// TIA Portal project "Bai 7" (V16)

(* hardware
DEVICE "S7-1200 station_1"  S7-1200 Station
   slot 0: "Rack_0"  S7-1200 Rack  Rack  V1.0
   slot 1: "PLC_1"  CPU 1214C DC/DC/DC  6ES7 214-1AG40-0XB0  V4.2
   slot 2: "DQ 16xRelay_1"  SM 1222 DQ16 x relay  6ES7 222-1HH32-0XB0  V2.0
*)

// ===== PLC "PLC_1"  CPU 1214C DC/DC/DC =====

VAR_GLOBAL   // PLC tag table "Default tag table"
   "Start" AT %I0.0 : Bool;
   "Quay_DC" AT %Q9.1 : Bool;
   "Khoan" AT %Q9.2 : Bool;
   "Biến giữ chương trình" AT %M0.0 : Bool;
   "SQ1" AT %I0.1 : Bool;
   "Biến giữ timer T5" AT %M1.1 : Bool;
   "Biến kích động cơ" AT %M1.2 : Bool;
   "Stop" AT %I1.0 : Bool;
   "Tag_11" AT %M1.3 : Bool;
   "Tag_12" AT %M0.1 : Bool;
   "Biến giữ quay DC" AT %M0.2 : Bool;
   "Tag_1" AT %M1.4 : Bool;
   "Tag_2" AT %M1.7 : Bool;
   "Tag_10" AT %M1.0 : Bool;
   "Biến kích nhánh 2" AT %M0.7 : Bool;
   "SQ2" AT %I0.2 : Bool;
   "SQ3" AT %I0.3 : Bool;
   "Biến giữ kẹp phôi" AT %M0.3 : Bool;
   "Biến giữ khoan" AT %M0.4 : Bool;
   "KepPhoi" AT %Q9.3 : Bool;
   "Biến giữ timer T3" AT %M0.5 : Bool;
   "Biến giữ timer T4" AT %M0.6 : Bool;
END_VAR

// folder: System blocks/Program resources

DATA_BLOCK "T1"   // DB1
{ S7_Optimized_Access := 'TRUE' }
AUTHOR : Simatic
FAMILY : IEC
NAME : IEC_TMR
VERSION : 1.0
// stored: InstanceOfName IEC_TIMER
"IEC_TIMER"
BEGIN
END_DATA_BLOCK

DATA_BLOCK "T2"   // DB2
{ S7_Optimized_Access := 'TRUE' }
AUTHOR : Simatic
FAMILY : IEC
NAME : IEC_TMR
VERSION : 1.0
// stored: InstanceOfName IEC_TIMER
"IEC_TIMER"
BEGIN
END_DATA_BLOCK

DATA_BLOCK "T3"   // DB3
{ S7_Optimized_Access := 'TRUE' }
AUTHOR : Simatic
FAMILY : IEC
NAME : IEC_TMR
VERSION : 1.0
// stored: InstanceOfName IEC_TIMER
"IEC_TIMER"
BEGIN
END_DATA_BLOCK

DATA_BLOCK "T4"   // DB4
{ S7_Optimized_Access := 'TRUE' }
AUTHOR : Simatic
FAMILY : IEC
NAME : IEC_TMR
VERSION : 1.0
// stored: InstanceOfName IEC_TIMER
"IEC_TIMER"
BEGIN
END_DATA_BLOCK

DATA_BLOCK "T5"   // DB5
{ S7_Optimized_Access := 'TRUE' }
AUTHOR : Simatic
FAMILY : IEC
NAME : IEC_TMR
VERSION : 1.0
// stored: InstanceOfName IEC_TIMER
"IEC_TIMER"
BEGIN
END_DATA_BLOCK

DATA_BLOCK "T6"   // DB6
{ S7_Optimized_Access := 'TRUE' }
AUTHOR : Simatic
FAMILY : IEC
NAME : IEC_TMR
VERSION : 1.0
// stored: InstanceOfName IEC_TIMER
"IEC_TIMER"
BEGIN
END_DATA_BLOCK

// folder: (top level)

ORGANIZATION_BLOCK "Main"   // OB1, LAD, ProgramCycle
TITLE = "Main Program Sweep (Cycle)"
{ S7_Optimized_Access := 'TRUE' }
VERSION : 0.1
   VAR_INPUT
      Initial_Call : Bool;   // Initial call of this OB
      Remanence : Bool;   // =True, if remanent data are available
   END_VAR
   VAR_TEMP   // added for the SCL form of the ladder/FBD networks
      _w1 : Bool;
   END_VAR
BEGIN

REGION Network 1
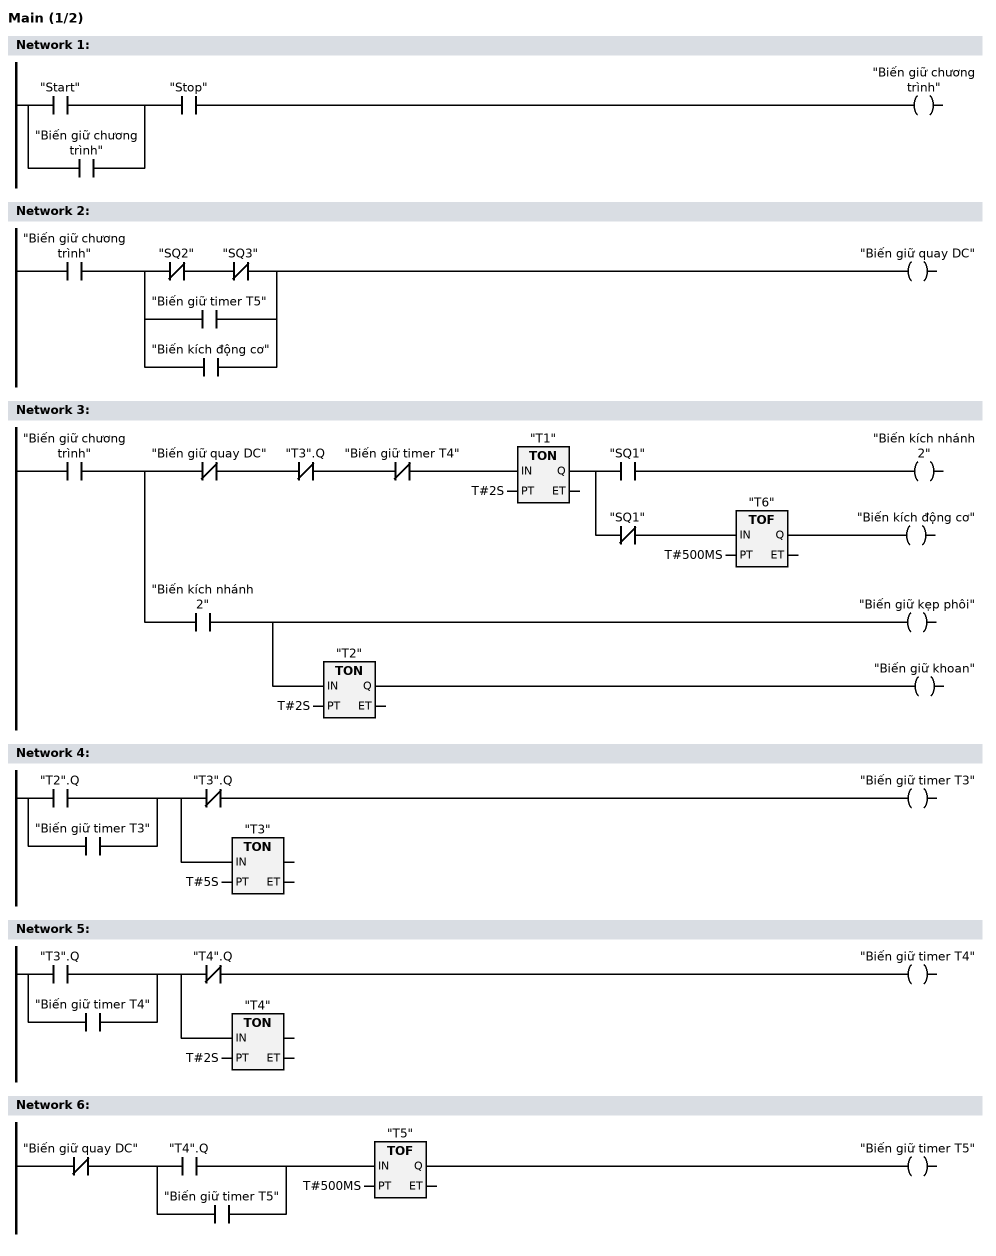
   RUNG wire#powerrail
      Contact( "Start" )
      wire#w1
      Contact( "Stop" )
      Coil( "Biến giữ chương trình" )
   END_RUNG
   RUNG wire#powerrail
      Contact( "Biến giữ chương trình" )
   END_RUNG wire#w1
   // the same network as SCL:
   "Biến giữ chương trình" := ("Start" OR "Biến giữ chương trình") AND "Stop";
END_REGION

REGION Network 2
   RUNG wire#powerrail
      Contact( "Biến giữ chương trình" )
      wire#w1
      I_Contact( "SQ2" )
      I_Contact( "SQ3" )
      wire#w2
      Coil( "Biến giữ quay DC" )
   END_RUNG
   RUNG wire#w1
      Contact( "Biến giữ timer T5" )
   END_RUNG wire#w2
   RUNG wire#w1
      Contact( "Biến kích động cơ" )
   END_RUNG wire#w2
   // the same network as SCL:
   "Biến giữ quay DC" := "Biến giữ chương trình" AND ((NOT "SQ2" AND NOT "SQ3") OR "Biến giữ timer T5" OR "Biến kích động cơ");
END_REGION

REGION Network 3
   "T1".TON(IN := "Biến giữ chương trình" AND NOT "Biến giữ quay DC" AND NOT "T3".Q AND NOT "Biến giữ timer T4",
            PT := T#2S);
   "Biến kích nhánh 2" := "T1".Q AND "SQ1";
   "T6".TOF(IN := "T1".Q AND NOT "SQ1", PT := T#500MS);
   "Biến kích động cơ" := "T6".Q;
   "Biến giữ kẹp phôi" := "Biến giữ chương trình" AND "Biến kích nhánh 2";
   "T2".TON(IN := "Biến giữ kẹp phôi", PT := T#2S);
   "Biến giữ khoan" := "T2".Q;
END_REGION

REGION Network 4
   #_w1 := "T2".Q OR "Biến giữ timer T3";
   "Biến giữ timer T3" := #_w1 AND NOT "T3".Q;
   "T3".TON(IN := #_w1, PT := T#5S);
END_REGION

REGION Network 5
   #_w1 := "T3".Q OR "Biến giữ timer T4";
   "Biến giữ timer T4" := #_w1 AND NOT "T4".Q;
   "T4".TON(IN := #_w1, PT := T#2S);
END_REGION

REGION Network 6
   "T5".TOF(IN := NOT "Biến giữ quay DC" AND ("T4".Q OR "Biến giữ timer T5"), PT := T#500MS);
   "Biến giữ timer T5" := "T5".Q;
END_REGION

REGION Network 7
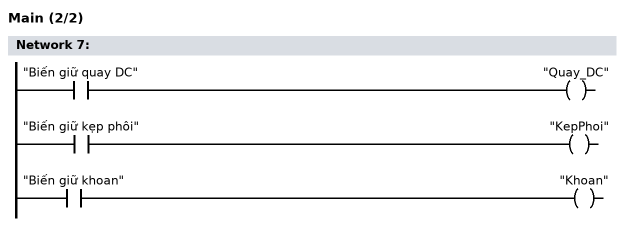
   RUNG wire#powerrail
      Contact( "Biến giữ quay DC" )
      Coil( "Quay_DC" )
   END_RUNG
   RUNG wire#powerrail
      Contact( "Biến giữ kẹp phôi" )
      Coil( "KepPhoi" )
   END_RUNG
   RUNG wire#powerrail
      Contact( "Biến giữ khoan" )
      Coil( "Khoan" )
   END_RUNG
   // the same network as SCL:
   "Quay_DC" := "Biến giữ quay DC";
   "KepPhoi" := "Biến giữ kẹp phôi";
   "Khoan" := "Biến giữ khoan";
END_REGION
END_ORGANIZATION_BLOCK